// TIA Portal V20 export
TYPE "InPut"
   STRUCT
      TrfInSetBegin : Bool;   // Command in from Graph / Load Begin: condition to start transfer IN set
      TrfInSetIntlkOk : Bool;   // Transfer IN Interlock Set OK
      TrfInResIntlkOk : Bool;   // Transfer IN Interlock Reset OKt
      TrfOutSetBegin : Bool;   // Unload Begin: condition to start transfer OUT set
      TrfOutSetIntlkOk : Bool;   // Transfer Out Interlock Set Ok
      TrfOutResIntlkOk : Bool;   // Transfer OUT Interlock Reset Ok
      TrfOutResBegin : Bool;
   END_STRUCT;
END_TYPE
